PROGRAM PRG_Gas_Selection
VAR
	
	CurrentGas: E_GasType;
	{attribute 'pytmc' := '
	pv: EM1K0:GMD:GAS_TYPE ;
	type: mbbi ;
	field: ZRST none ;
	field: ONST Neon;
	field: TWST Argon ;
	field: THST Krypton ;
	field: FRST Xenon ;
	io: i
	'}
	SelectedGas: E_GasType;
END_VAR

(* Gas selection includes a purge and checks interlocks*)

if ( VVC_83.iq_stValve.q_xOPN_DO) then
	CurrentGas := E_GasType.Neon;
	elsif ( VVC_84.iq_stValve.q_xOPN_DO) then
		CurrentGas := E_GasType.Argon;
		elsif ( VVC_85.iq_stValve.q_xOPN_DO) then
		CurrentGas := E_GasType.Krypton;
			elsif ( VVC_86.iq_stValve.q_xOPN_DO) then
			CurrentGas := E_GasType.Xenon;
			 else 
				 CurrentGas := E_GasType.none;
END_IF


If( CurrentGas <> SelectedGas) AND NOT (CurrentGas=E_GasType.none) then
	bStartPurge_sw := true;
END_IF

if NOT(bStartPurge_sw) AND(bPurgeDone) then
	case SelectedGas of
	E_GasType.none: // all valves closed
		VVC_83.M_Set_OPN_SW(false);
		VVC_84.M_Set_OPN_SW(false);
		VVC_85.M_Set_OPN_SW(false);
		VVC_86.M_Set_OPN_SW(false);
	E_GasType.Neon:
		VVC_83.M_Set_OPN_SW(TRUE);
		VVC_84.M_Set_OPN_SW(false);
		VVC_85.M_Set_OPN_SW(false);
		VVC_86.M_Set_OPN_SW(false);
	E_GasType.Argon: 
		VVC_83.M_Set_OPN_SW(false);
		VVC_84.M_Set_OPN_SW(TRUE);
		VVC_85.M_Set_OPN_SW(false);
		VVC_86.M_Set_OPN_SW(false); 
	E_GasType.Krypton: 
		VVC_83.M_Set_OPN_SW(false);
		VVC_84.M_Set_OPN_SW(false);
		VVC_85.M_Set_OPN_SW(TRUE);
		VVC_86.M_Set_OPN_SW(false);
	E_GasType.Xenon: 
		VVC_83.M_Set_OPN_SW(false);
		VVC_84.M_Set_OPN_SW(false);
		VVC_85.M_Set_OPN_SW(false);
		VVC_86.M_Set_OPN_SW(TRUE);
	END_CASE
END_IF


/// vcn and vgp on manual or auto??

END_PROGRAM

(* stored: Version 1.1.0.1, ProductVersion 3.1.4022.18
   POU PRG_Gas_Selection: Id {f65eb335-21e5-43a7-a5c6-4b463c324e82}, SpecialFunc None *)
